{attribute 'qualified_only'}
{attribute 'strict'}
TYPE E_ConveyorMode :
(
    IDLE              := 0,
    RUNNING_FORWARD   := 10,
    RUNNING_BACKWARD  := 20,
    FAULT             := 99
);
END_TYPE

(* stored: Version 1.1.0.1, ProductVersion 3.1.4024.16
   DUT E_ConveyorMode: Id {e2a1b3c4-d5e6-7890-abcd-ef1234567890} *)
